// TIA Portal project "PLC_AGV.CENTRAL_V15" (V15)

(* hardware
DEVICE "ET 200S station_1"  ET 200S station
   slot 0: "Rack_0"  Rail
   slot 2: "PLC_AGV.CENTRAL"  IM151-8 PN/DP CPU  6ES7 151-8AB01-0AB0  V3.2
      slot 1: "PROFINET interface_1"  PN-IO
         slot 1: "Port_1"  Port
         slot 2: "Port_2"  Port
         slot 3: "Port_3"  Port
   slot 4: "PM-E 24VDC_1"  PM-E 24VDC  6ES7 138-4CA01-0AA0
   slot 5: "8DI x 24VDC_1"  8DI x 24VDC  6ES7 131-4BF00-0AA0
   slot 6: "8DI x 24VDC_2"  8DI x 24VDC  6ES7 131-4BF00-0AA0
   slot 7: "8DI x 24VDC_3"  8DI x 24VDC  6ES7 131-4BF00-0AA0
   slot 8: "8DI x 24VDC_4"  8DI x 24VDC  6ES7 131-4BF00-0AA0
   slot 9: "8DO x 24VDC / 0.5A_1"  8DO x 24VDC / 0.5A  6ES7 132-4BF00-0AA0
   slot 10: "8DO x 24VDC / 0.5A_2"  8DO x 24VDC / 0.5A  6ES7 132-4BF00-0AA0
   slot 11: "8DO x 24VDC / 0.5A_3"  8DO x 24VDC / 0.5A  6ES7 132-4BF00-0AA0
   slot 12: "8DO x 24VDC / 0.5A_4"  8DO x 24VDC / 0.5A  6ES7 132-4BF00-0AA0
*)

// ===== PLC "PLC_AGV.CENTRAL"  IM151-8 PN/DP CPU =====

VAR_GLOBAL   // PLC tag table "Default tag table"
   "HORN" AT %Q5.0 : Bool;
   "LAMP1" AT %Q5.2 : Bool;
   "LAMP2" AT %Q5.4 : Bool;
   "LAMP3" AT %Q5.6 : Bool;
   "DI.Start_D1" AT %I3.0 : Bool;
   "DI.Stop_D1" AT %I3.1 : Bool;
   "DI.Start_D2" AT %I3.2 : Bool;
   "DI.Stop_D2" AT %I3.3 : Bool;
   "DI.Start_D3" AT %I3.4 : Bool;
   "DI.Stop_D3" AT %I3.5 : Bool;
   "DI.Start_D4" AT %I3.6 : Bool;
   "DI.Stop_D4" AT %I3.7 : Bool;
   "DI_BufferScanner" AT %I4.0 : Bool;   // Scanner to check buffer height
   "DO_GreenLight" AT %Q6.0 : Bool;   // Green light to indicate buffer height
   "DO_RedLight" AT %Q6.1 : Bool;   // Red light - buffer overheight
   "DO_BufferBuzzer" AT %Q6.2 : Bool;   // Buzzer buffer overheight
   "Always_True" AT %M10.0 : Bool;
   "Always_False" AT %M10.1 : Bool;
END_VAR

VAR_GLOBAL CONSTANT   // PLC tag table "Default tag table"
   "QTY.AGV" : Int := 7;
   "MAX.STATIONS" : Int := 8;
END_VAR

VAR_GLOBAL   // PLC tag table "ClockMemory"
   "CM_0.1s" AT %M0.0 : Bool;
   "CM_0.2s" AT %M0.1 : Bool;
   "CM_0.4s" AT %M0.2 : Bool;
   "CM_0.5s" AT %M0.3 : Bool;
   "CM_0.8s" AT %M0.4 : Bool;
   "CM_1s" AT %M0.5 : Bool;
   "CM_1.6s" AT %M0.6 : Bool;
   "CM_2s" AT %M0.7 : Bool;
END_VAR

VAR_GLOBAL   // PLC tag table "IO tag table"
   "STATION1.STOP" AT %I1.0 : Bool;
   "STATION1.RUN" AT %I1.1 : Bool;
   "STATION2.STOP" AT %I1.2 : Bool;
   "STATION2.RUN" AT %I1.3 : Bool;
   "STATION3.STOP" AT %I1.4 : Bool;
   "STATION3.RUN" AT %I1.5 : Bool;
   "STATION4.STOP" AT %I1.6 : Bool;
   "STATION4.RUN" AT %I1.7 : Bool;
   "STATION5.STOP" AT %I2.0 : Bool;
   "STATION5.RUN" AT %I2.1 : Bool;
   "STATION6.STOP" AT %I2.2 : Bool;
   "STATION6.RUN" AT %I2.3 : Bool;
END_VAR

VAR_GLOBAL   // PLC tag table "MemoriasTakt"
   "Me_PararLinha" AT %M20.0 : Bool;
   "Me_Emergencia" AT %M20.1 : Bool;
   "Me_EmTurno" AT %M20.2 : Bool;
   "Me_ResetTakt" AT %M20.3 : Bool;
   "Me_ParadaProgramada" AT %M20.4 : Bool;
   "Me_PararLinhaAgv" AT %M20.5 : Bool;
   "Ret_Val" AT %MW2 : Int;
   "Error" AT %M1.0 : Bool;
   "Statuts" AT %MW4 : Word;
   "C_Conect" AT %M1.1 : Bool;
   "C_Status" AT %MW6 : Word;
END_VAR

TYPE "Agv.Database"
   STRUCT
      Emergencia : Bool;   // Botao de Emergecencia
      Warning : Bool;   // Area de Warning do Scanner
      Safety : Bool;   // Area de Safety do Scanner
      ConectarTakt : Bool;   // 0 - Desconectado / 1 - Conectado
      Rodando : Bool;
      Falha : Bool;
      AutomaticoManual : Byte;   // 1 - Manual / 2 - Automatico
      VelocidadeAtual : Int;   // Velocidade Atual
      Posto : Byte;   // Posto em que o AGV está
      Comando : Byte;   // Ultimo comando
      Velocidade : Byte;   // Velocidade Setada
      Processo : Byte;   // 1 - Ecu / 2 - SKD
      "Erros.Agv" : Byte;   // 0 á 256, cada numero um erro. 1 - Tudo Ok
      "Erros.Pgv" : Byte;   // 0 á 256, cada numero um erro. 1 - Tudo Ok
      "Erros.Rfid" : Byte;   // 0 á 256, cada numero um erro. 1 - Tudo Ok
      "Erros.MotorPasso" : Byte;   // 0 á 256, cada numero um erro. 1 - Tudo Ok
      "Erros.IOLink" : Byte;   // 0 á 256, cada numero um erro. 1 - Tudo Ok
      "Erros.Comunicacao" : Byte;   // 0 á 256, cada numero um erro. 1 - Tudo Ok
      Reservado : Byte;   // Reservado
      Reservado_1 : Byte;   // Reservado
      Reservado_2 : Byte;   // Reservado
      Reservado_3 : Byte;   // Reservado
      Reservado_4 : Byte;   // Reservado
      Reservado_5 : Byte;   // Reservado
      Reservado_6 : Byte;   // Reservado
      Reservado_7 : Byte;   // Reservado
      Reservado_8 : Byte;   // Reservado
   END_STRUCT;
END_TYPE

TYPE "Takt.Database"
   STRUCT
      EmergenciaECU : Bool;   // Emergencia
      EmergenciaSKD : Bool;   // Emergencia
      StartAgvECU : Bool;   // Start by takt
      StopAgvECU : Bool;   // Stop by takt
      StartAgvSKD : Bool;   // Start by takt
      StopAgvSKD : Bool;   // Stop by takt
      WatchDog : Bool;   // WatchDog
      TOD : Time_Of_Day;   // Time of day
   END_STRUCT;
END_TYPE

TYPE "Scada.Datebase"
   STRUCT
      Turnos : Struct
         Inicio : Array[0..2] of Time_Of_Day;
         Fim : Array[0..2] of Time_Of_Day;
      END_STRUCT;
      Paradas_Programadas : Struct
         Inicio : Array[0..5] of Time_Of_Day;
         Fim : Array[0..5] of Time_Of_Day;
      END_STRUCT;
      Dias_Da_Semana : Array[0..6] of Bool;
      ParametrosTakt : Array[0..2] of Struct
         Tempo_Takt : Int;
         ObjetivoTurno : Int;
      END_STRUCT;
      DiaDaSemana : Int;
   END_STRUCT;
   // // Dias_Da_Semana[0] : Segunda-Feira
   // // Dias_Da_Semana[1] : Terça-Feira
   // // Dias_Da_Semana[2] : Quarta-Feira
   // // Dias_Da_Semana[3] : Quinta-Feira
   // // Dias_Da_Semana[4] : Sexta-Feira
   // // Dias_Da_Semana[5] : Sabado
   // // Dias_Da_Semana[6] : Domingo
   // // ParametrosTakt[0] : Parametros do Takt do 1 turno
   // // ParametrosTakt[1] : Parametros do Takt do 2 turno
   // // ParametrosTakt[2] : Parametros do Takt do 3 turno
   // // Turnos.Inicio[0] : Incio 1 Turno
   // // Turnos.Inicio[1] : Incio 2 Turno
   // // Turnos.Inicio[2] : Incio 3 Turno
   // // Turnos.Fim[0] : Fim 1 Turno
   // // Turnos.Fim[1] : Fim 2 Turno
   // // Turnos.Fim[2] : Fim 3 Turno
   // // Paradas_Programadas.Inicio[0] : Inicio Parada Programada 1
   // // Paradas_Programadas.Inicio[1] : Inicio Parada Programada 2
   // // Paradas_Programadas.Fim[0] : Fim Parada Programada 1
   // // Paradas_Programadas.Inicio[2] : Inicio Parada Programada 3
   // // Paradas_Programadas.Inicio[3] : Inicio Parada Programada 4
   // // Paradas_Programadas.Inicio[4] : Inicio Parada Programada 5
   // // Paradas_Programadas.Inicio[5] : Inicio Parada Programada 6
   // // Paradas_Programadas.Fim[1] : Fim Parada Programada 2
   // // Paradas_Programadas.Fim[2] : Fim Parada Programada 3
   // // Paradas_Programadas.Fim[3] : Fim Parada Programada 4
   // // Paradas_Programadas.Fim[4] : Fim Parada Programada 5
   // // Paradas_Programadas.Fim[5] : Fim Parada Programada 6
END_TYPE

TYPE "UltimasParadas"
   STRUCT
      NumeroPosto : Int;
      InicioParada : Time_Of_Day;
      FimParada : Time_Of_Day;
      DiaDaParada : Date;
   END_STRUCT;
END_TYPE

TYPE "Central.Database"
   STRUCT
      Dados_Agv : Array[0..12] of "Agv.Database";
      Dados_Takt : Struct
         Tempo_Takt : DInt;
         Tempo_StopTime : DInt;
         Objetivo : Int;
         Atual : Int;
         TempoParada : DInt;
         Andons : Array[0..8] of Bool;
      END_STRUCT;
      Dados_Paradas : Array[0..20] of "UltimasParadas";
   END_STRUCT;
END_TYPE

// folder: 01_Takt/02_DB

DATA_BLOCK "DB100_LogicaTaktEcu"   // DB100
{ S7_Optimized_Access := 'FALSE' }
AUTHOR : ssbjvq
VERSION : 0.1
// stored: InstanceOfName FB100_LogicaTaktEcu
"FB100_LogicaTaktEcu"
BEGIN
END_DATA_BLOCK

DATA_BLOCK "DB101_SinaisEmTurno"   // DB101
{ S7_Optimized_Access := 'FALSE' }
VERSION : 0.1
// stored: InstanceOfName FB101_SinaisEmTurno
"FB101_SinaisEmTurno"
BEGIN
END_DATA_BLOCK

DATA_BLOCK "DB102_SinaisDeAndons"   // DB102
{ S7_Optimized_Access := 'FALSE' }
VERSION : 0.1
// stored: InstanceOfName FB102_SinaisDeAndons
"FB102_SinaisDeAndons"
BEGIN
END_DATA_BLOCK

DATA_BLOCK "DB103_AndonsAgvs"   // DB103
{ S7_Optimized_Access := 'FALSE' }
VERSION : 0.1
// stored: InstanceOfName FB103_AndonsAgvs
"FB103_AndonsAgvs"
BEGIN
END_DATA_BLOCK

// folder: 02_Comunicação/02_DB

DATA_BLOCK "DB200_TaktToAgv"   // DB200
TITLE = DB1_TaktToAgv
{ S7_Optimized_Access := 'FALSE' }
AUTHOR : ssbjvq
VERSION : 0.1
// DB1_TaktToAgv
   VAR
      Dados : "Takt.Database";
   END_VAR
BEGIN
   Dados.WatchDog := TRUE;
END_DATA_BLOCK

DATA_BLOCK "DB201_Comunicação"   // DB201
{ S7_Optimized_Access := 'FALSE' }
AUTHOR : ssbjvq
VERSION : 0.1
// stored: InstanceOfName FB201_Comunicação
"FB201_Comunicação"
BEGIN
END_DATA_BLOCK

// folder: 03_Scada

DATA_BLOCK "DB300_ScadaToCentral"   // DB300
TITLE = DB300_MestreToCentral
{ S7_Optimized_Access := 'FALSE' }
VERSION : 0.1
// DB300_MestreToCentral
   VAR
      Data : "Scada.Datebase";
   END_VAR
BEGIN
   Data.Turnos.Inicio[0] := TOD#08:00:00;
   Data.Turnos.Inicio[1] := TOD#00:00:00;
   Data.Turnos.Inicio[2] := TOD#00:00:00;
   Data.Turnos.Fim[0] := TOD#15:55:00;
   Data.Turnos.Fim[1] := TOD#00:00:00;
   Data.Turnos.Fim[2] := TOD#00:00:00;
   Data.Dias_Da_Semana[0] := TRUE;
   Data.Dias_Da_Semana[1] := TRUE;
   Data.Dias_Da_Semana[2] := TRUE;
   Data.Dias_Da_Semana[3] := TRUE;
   Data.Dias_Da_Semana[4] := TRUE;
   Data.ParametrosTakt[0].Tempo_Takt := 600;
   Data.ParametrosTakt[0].ObjetivoTurno := 48;
   Data.ParametrosTakt[1].Tempo_Takt := 600;
   Data.ParametrosTakt[1].ObjetivoTurno := 48;
   Data.ParametrosTakt[2].Tempo_Takt := 600;
   Data.ParametrosTakt[2].ObjetivoTurno := 48;
   Data.DiaDaSemana := 2;
   Data.Paradas_Programadas.Fim[0] := TOD#12:15:00;
   Data.Paradas_Programadas.Inicio[0] := TOD#11:15:00;
END_DATA_BLOCK

DATA_BLOCK "DB301_CentralToScada"   // DB301
TITLE = DB301_CentralToScada
{ S7_Optimized_Access := 'FALSE' }
VERSION : 0.1
// DB301_CentralToScada
   VAR
      Data : "Central.Database";
   END_VAR
BEGIN
END_DATA_BLOCK

// folder: 04_Services/02_DB

DATA_BLOCK "FB1000_Clock_DB"   // DB1
{ S7_Optimized_Access := 'FALSE' }
VERSION : 0.1
// stored: InstanceOfName FB1000_Clock
"FB1000_Clock"
BEGIN
END_DATA_BLOCK

// folder: (top level)

ORGANIZATION_BLOCK "Main"   // OB1, LAD
TITLE = "Main Program Sweep (Cycle)"
{ S7_Optimized_Access := 'FALSE' }
VERSION : 0.1
   VAR_TEMP
      OB1_EV_CLASS : Byte;   // Bits 0-3 = 1 (Coming event), Bits 4-7 = 1 (Event class 1)
      OB1_SCAN_1 : Byte;   // 1 (Cold restart scan 1 of OB 1), 3 (Scan 2-n of OB 1)
      OB1_PRIORITY : Byte;   // Priority of OB Execution
      OB1_OB_NUMBR : Byte;   // 1 (Organization block 1, OB1)
      OB1_RESERVED_1 : Byte;   // Reserved for system
      OB1_RESERVED_2 : Byte;   // Reserved for system
      OB1_PREV_CYCLE : Int;   // Cycle time of previous OB1 scan (milliseconds)
      OB1_MIN_CYCLE : Int;   // Minimum cycle time of OB1 (milliseconds)
      OB1_MAX_CYCLE : Int;   // Maximum cycle time of OB1 (milliseconds)
      OB1_DATE_TIME : Date_And_Time;   // Date and time OB1 started
   END_VAR
BEGIN

REGION Network 1: Filtro dos botões de Andon
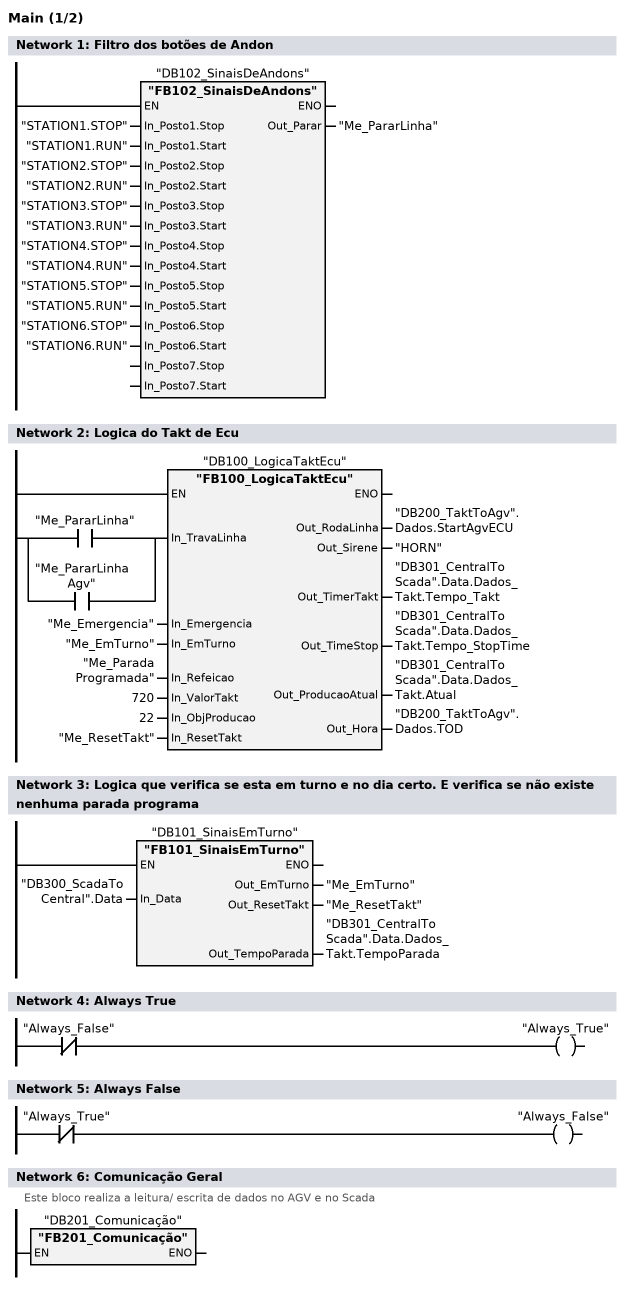
   RUNG wire#powerrail
      "DB102_SinaisDeAndons"("In_Posto1.Stop" := "STATION1.STOP", "In_Posto1.Start" := "STATION1.RUN", "In_Posto2.Stop" := "STATION2.STOP", "In_Posto2.Start" := "STATION2.RUN", "In_Posto3.Stop" := "STATION3.STOP", "In_Posto3.Start" := "STATION3.RUN", "In_Posto4.Stop" := "STATION4.STOP", "In_Posto4.Start" := "STATION4.RUN", "In_Posto5.Stop" := "STATION5.STOP", "In_Posto5.Start" := "STATION5.RUN", "In_Posto6.Stop" := "STATION6.STOP", "In_Posto6.Start" := "STATION6.RUN", "In_Posto7.Stop" :=, "In_Posto7.Start" :=, Out_Parar => "Me_PararLinha")
   END_RUNG
   // the same network as SCL:
   "DB102_SinaisDeAndons"("In_Posto1.Stop" := "STATION1.STOP",   // "FB102_SinaisDeAndons"
                          "In_Posto1.Start" := "STATION1.RUN",
                          "In_Posto2.Stop" := "STATION2.STOP",
                          "In_Posto2.Start" := "STATION2.RUN",
                          "In_Posto3.Stop" := "STATION3.STOP",
                          "In_Posto3.Start" := "STATION3.RUN",
                          "In_Posto4.Stop" := "STATION4.STOP",
                          "In_Posto4.Start" := "STATION4.RUN",
                          "In_Posto5.Stop" := "STATION5.STOP",
                          "In_Posto5.Start" := "STATION5.RUN",
                          "In_Posto6.Stop" := "STATION6.STOP",
                          "In_Posto6.Start" := "STATION6.RUN",
                          Out_Parar => "Me_PararLinha");
END_REGION

REGION Network 2: Logica do Takt de Ecu
   RUNG wire#powerrail
      "DB100_LogicaTaktEcu"(In_TravaLinha := wire#w1, In_Emergencia := "Me_Emergencia", In_EmTurno := "Me_EmTurno", In_Refeicao := "Me_ParadaProgramada", In_ValorTakt := 720, In_ObjProducao := 22, In_ResetTakt := "Me_ResetTakt", Out_RodaLinha => "DB200_TaktToAgv".Dados.StartAgvECU, Out_Sirene => "HORN", Out_TimerTakt => "DB301_CentralToScada".Data.Dados_Takt.Tempo_Takt, Out_TimeStop => "DB301_CentralToScada".Data.Dados_Takt.Tempo_StopTime, Out_ProducaoAtual => "DB301_CentralToScada".Data.Dados_Takt.Atual, Out_Hora => "DB200_TaktToAgv".Dados.TOD)
   END_RUNG
   RUNG wire#powerrail
      Contact( "Me_PararLinha" )
   END_RUNG wire#w1
   RUNG wire#powerrail
      Contact( "Me_PararLinhaAgv" )
   END_RUNG wire#w1
   // the same network as SCL:
   "DB100_LogicaTaktEcu"(In_TravaLinha := "Me_PararLinha" OR "Me_PararLinhaAgv",   // "FB100_LogicaTaktEcu"
                         In_Emergencia := "Me_Emergencia",
                         In_EmTurno := "Me_EmTurno",
                         In_Refeicao := "Me_ParadaProgramada",
                         In_ValorTakt := 720,
                         In_ObjProducao := 22,
                         In_ResetTakt := "Me_ResetTakt",
                         Out_RodaLinha => "DB200_TaktToAgv".Dados.StartAgvECU,
                         Out_Sirene => "HORN",
                         Out_TimerTakt => "DB301_CentralToScada".Data.Dados_Takt.Tempo_Takt,
                         Out_TimeStop => "DB301_CentralToScada".Data.Dados_Takt.Tempo_StopTime,
                         Out_ProducaoAtual => "DB301_CentralToScada".Data.Dados_Takt.Atual,
                         Out_Hora => "DB200_TaktToAgv".Dados.TOD);
END_REGION

REGION Network 3: Logica que verifica se esta em turno e no dia certo. E verifica se não existe nenhuma parada programa
   RUNG wire#powerrail
      "DB101_SinaisEmTurno"(In_Data := "DB300_ScadaToCentral".Data, Out_EmTurno => "Me_EmTurno", Out_ResetTakt => "Me_ResetTakt", Out_TempoParada => "DB301_CentralToScada".Data.Dados_Takt.TempoParada)
   END_RUNG
   // the same network as SCL:
   "DB101_SinaisEmTurno"(In_Data := "DB300_ScadaToCentral".Data,   // "FB101_SinaisEmTurno"
                         Out_EmTurno => "Me_EmTurno",
                         Out_ResetTakt => "Me_ResetTakt",
                         Out_TempoParada => "DB301_CentralToScada".Data.Dados_Takt.TempoParada);
END_REGION

REGION Network 4: Always True
   RUNG wire#powerrail
      I_Contact( "Always_False" )
      Coil( "Always_True" )
   END_RUNG
   // the same network as SCL:
   "Always_True" := NOT "Always_False";
END_REGION

REGION Network 5: Always False
   RUNG wire#powerrail
      I_Contact( "Always_True" )
      Coil( "Always_False" )
   END_RUNG
   // the same network as SCL:
   "Always_False" := NOT "Always_True";
END_REGION

REGION Network 6: Comunicação Geral
   // Este bloco realiza a leitura/ escrita de dados no AGV e no Scada
   RUNG wire#powerrail
      "DB201_Comunicação"()
   END_RUNG
   // the same network as SCL:
   "DB201_Comunicação"();   // "FB201_Comunicação"
END_REGION

REGION Network 7: Sinais de Andon dos Agvs
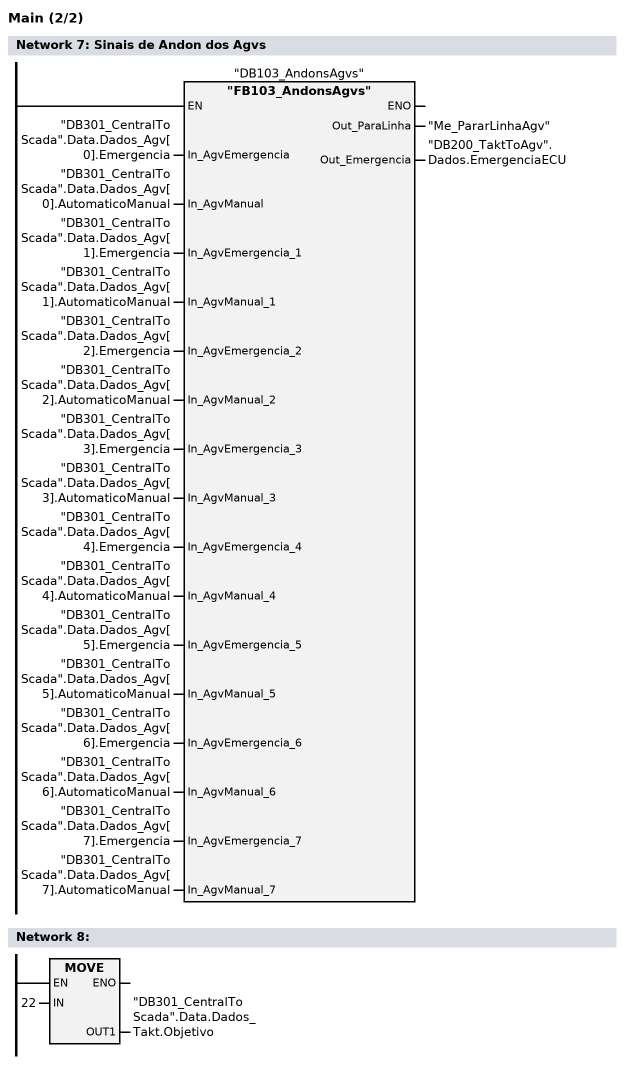
   RUNG wire#powerrail
      "DB103_AndonsAgvs"(In_AgvEmergencia := "DB301_CentralToScada".Data.Dados_Agv[0].Emergencia, In_AgvManual := "DB301_CentralToScada".Data.Dados_Agv[0].AutomaticoManual, In_AgvEmergencia_1 := "DB301_CentralToScada".Data.Dados_Agv[1].Emergencia, In_AgvManual_1 := "DB301_CentralToScada".Data.Dados_Agv[1].AutomaticoManual, In_AgvEmergencia_2 := "DB301_CentralToScada".Data.Dados_Agv[2].Emergencia, In_AgvManual_2 := "DB301_CentralToScada".Data.Dados_Agv[2].AutomaticoManual, In_AgvEmergencia_3 := "DB301_CentralToScada".Data.Dados_Agv[3].Emergencia, In_AgvManual_3 := "DB301_CentralToScada".Data.Dados_Agv[3].AutomaticoManual, In_AgvEmergencia_4 := "DB301_CentralToScada".Data.Dados_Agv[4].Emergencia, In_AgvManual_4 := "DB301_CentralToScada".Data.Dados_Agv[4].AutomaticoManual, In_AgvEmergencia_5 := "DB301_CentralToScada".Data.Dados_Agv[5].Emergencia, In_AgvManual_5 := "DB301_CentralToScada".Data.Dados_Agv[5].AutomaticoManual, In_AgvEmergencia_6 := "DB301_CentralToScada".Data.Dados_Agv[6].Emergencia, In_AgvManual_6 := "DB301_CentralToScada".Data.Dados_Agv[6].AutomaticoManual, In_AgvEmergencia_7 := "DB301_CentralToScada".Data.Dados_Agv[7].Emergencia, In_AgvManual_7 := "DB301_CentralToScada".Data.Dados_Agv[7].AutomaticoManual, Out_ParaLinha => "Me_PararLinhaAgv", Out_Emergencia => "DB200_TaktToAgv".Dados.EmergenciaECU)
   END_RUNG
   // the same network as SCL:
   "DB103_AndonsAgvs"(In_AgvEmergencia := "DB301_CentralToScada".Data.Dados_Agv[0].Emergencia,   // "FB103_AndonsAgvs"
                      In_AgvManual := "DB301_CentralToScada".Data.Dados_Agv[0].AutomaticoManual,
                      In_AgvEmergencia_1 := "DB301_CentralToScada".Data.Dados_Agv[1].Emergencia,
                      In_AgvManual_1 := "DB301_CentralToScada".Data.Dados_Agv[1].AutomaticoManual,
                      In_AgvEmergencia_2 := "DB301_CentralToScada".Data.Dados_Agv[2].Emergencia,
                      In_AgvManual_2 := "DB301_CentralToScada".Data.Dados_Agv[2].AutomaticoManual,
                      In_AgvEmergencia_3 := "DB301_CentralToScada".Data.Dados_Agv[3].Emergencia,
                      In_AgvManual_3 := "DB301_CentralToScada".Data.Dados_Agv[3].AutomaticoManual,
                      In_AgvEmergencia_4 := "DB301_CentralToScada".Data.Dados_Agv[4].Emergencia,
                      In_AgvManual_4 := "DB301_CentralToScada".Data.Dados_Agv[4].AutomaticoManual,
                      In_AgvEmergencia_5 := "DB301_CentralToScada".Data.Dados_Agv[5].Emergencia,
                      In_AgvManual_5 := "DB301_CentralToScada".Data.Dados_Agv[5].AutomaticoManual,
                      In_AgvEmergencia_6 := "DB301_CentralToScada".Data.Dados_Agv[6].Emergencia,
                      In_AgvManual_6 := "DB301_CentralToScada".Data.Dados_Agv[6].AutomaticoManual,
                      In_AgvEmergencia_7 := "DB301_CentralToScada".Data.Dados_Agv[7].Emergencia,
                      In_AgvManual_7 := "DB301_CentralToScada".Data.Dados_Agv[7].AutomaticoManual,
                      Out_ParaLinha => "Me_PararLinhaAgv",
                      Out_Emergencia => "DB200_TaktToAgv".Dados.EmergenciaECU);
END_REGION

REGION Network 8
   RUNG wire#powerrail
      { S7_GenerateENO := "TRUE" } Move(in := 22, out1 => "DB301_CentralToScada".Data.Dados_Takt.Objetivo)
   END_RUNG
   // the same network as SCL:
   "DB301_CentralToScada".Data.Dados_Takt.Objetivo := 22;
END_REGION
END_ORGANIZATION_BLOCK

// folder: 01_Takt/01_FB

FUNCTION_BLOCK "FB100_LogicaTaktEcu"   // FB100, SCL
TITLE = FB100_LogicaTaktEcu
{ S7_Optimized_Access := 'FALSE' }
AUTHOR : ssbjvq
VERSION : 0.1
// FB100_LogicaTaktEcu
   VAR_INPUT
      In_TravaLinha : Bool;   // Input dos andons. True - Para Linha/ False - Tudo Ok!
      In_Emergencia : Bool;   // Inout de Emergencia. True - Acionado/ False - Desacionado
      In_EmTurno : Bool;   // Input dos Em turno. True - Linha em turno/ False - Fora do turno
      In_Refeicao : Bool;   // Input de Pause Programada. True - Em horario de parada / False - Fora do horario de parada
      In_ValorTakt : Int;   // Input do valor do Takt
      In_ObjProducao : Int;   // Input do Objetivo de producao
      In_ResetTakt : Bool;   // Sinal que reseta o Stop Time
   END_VAR
   VAR_OUTPUT
      Out_RodaLinha : Bool;   // Out Roda Linha
      Out_Sirene : Bool;   // Out Sirene
      Out_TimerTakt : DInt;   // Out Tempo Takt
      Out_TimeStop : DInt;   // Out Tempo Stop time
      Out_ProducaoAtual : Int;   // Out Contagem Producao
      Out_Hora : Time_Of_Day;
   END_VAR
   VAR
      S_TudoOk : Bool;   // Inicia a contagem do Takt
      S_ResetTakt : Bool;   // Reseta o Takt
      S_StopLinha : Bool;   // Inicia a contagem do Stop time
      S_Reset_Stop : Bool;   // Reseta o Stop Time E Contagem Producao
      S_TaktTimeAtual : DInt;   // Tempo Atual do Takt ( Regressivo)
      Contador_Takt : CTU;   // Contador do Takt
      Contador_StopTime : CTU;   // Contador do Stop Time
      Contador_Producao : CTU;   // Contador de Producao
      Start_Takt : TP;
      S_DateTime : Date_And_Time;
      S_ResetAllTakt : Bool;
   END_VAR
   VAR_TEMP
      Err : Int;
   END_VAR
BEGIN
   (*
    BLOCO DESENVOLVIDO POR SSBJVQ R.4946
    BLOCO DO TAKT
   *)

   REGION Logica Takt
       IF #In_ResetTakt THEN
           #S_ResetTakt := 1;
           #S_TudoOk := 0;
           #S_StopLinha := 0;
           #S_ResetTakt := 0;
           #S_Reset_Stop := 1;
       END_IF;
       // Verifica as condições para acionar a contagem do Takt
       IF (#In_EmTurno AND NOT #In_Refeicao AND
           (#Contador_Takt.CV < #In_ValorTakt) AND (#Contador_Producao.CV < #In_ObjProducao)) AND NOT #In_ResetTakt THEN
           #S_TudoOk := 1;
           #S_StopLinha := 0;
           #S_ResetTakt := 0;
           #S_Reset_Stop := 0;

           // Verifica as condições para acionar a contagem do Stop Time
       ELSIF ((#In_Emergencia OR #In_TravaLinha) AND (#Contador_Takt.CV = #In_ValorTakt)
           AND (#Contador_Producao.CV < #In_ObjProducao) AND #In_EmTurno) AND NOT #In_ResetTakt THEN
           #S_TudoOk := 0;
           #S_StopLinha := 1;
           #S_ResetTakt := 0;
           #S_Reset_Stop := 0;
           // Verifica as condições para acionar o Reset Takt
       ELSIF (#In_EmTurno
           AND NOT #In_Refeicao AND NOT #In_Emergencia
           AND NOT #In_TravaLinha AND (#Contador_Takt.CV = #In_ValorTakt) AND #Contador_Takt.Q)AND NOT #In_ResetTakt THEN
           #S_ResetTakt := 1;
           // Verifica se esta em parada programada
       ELSIF NOT #In_EmTurno AND #In_Refeicao AND NOT #In_ResetTakt THEN
           #S_TudoOk := 0;
           #S_StopLinha := 0;
           #S_Reset_Stop := 0;
           #S_ResetTakt := 0;
       // Verifica as condições para acionar o Reset Stop Time
       ELSIF #In_ResetTakt THEN
           #S_Reset_Stop := 1;
           #S_TudoOk := 0;
           #S_StopLinha := 0;
           #S_ResetTakt := 1;
       ELSE
           #S_TudoOk := 0;
           #S_StopLinha := 0;
           #S_Reset_Stop := 0;
           #S_ResetTakt := 0;
       END_IF;

       #Err := RD_SYS_T(#S_DateTime);
   END_REGION

   IF DT_TO_TOD(#S_DateTime) >= TOD#07:00:00 AND  DT_TO_TOD(#S_DateTime)<= TOD#07:01:00
       OR DT_TO_TOD(#S_DateTime) >= TOD#17:00:00 AND  DT_TO_TOD(#S_DateTime)<= TOD#17:01:00
       OR DT_TO_TOD(#S_DateTime) >= TOD#00:00:00 AND  DT_TO_TOD(#S_DateTime)<= TOD#00:01:00 THEN
       #S_ResetAllTakt := 1;
   ELSE
       #S_ResetAllTakt := 0;
   END_IF;


   // Contém os contadores do TAKT, Stop Time e Producao
   REGION Contadores

       #Contador_Takt(CU := #S_TudoOk AND "CM_1s",
                      R := #S_ResetTakt OR #In_ResetTakt OR #S_ResetAllTakt ,
                      PV := #In_ValorTakt);
       #Contador_StopTime(CU := #S_StopLinha AND "CM_1s" ,
                          R :=  #S_Reset_Stop OR #In_ResetTakt OR #S_ResetAllTakt
                          ,
                          PV := 32747);
       #Contador_Producao(CU := #Contador_Takt.Q ,
                          R := #S_Reset_Stop OR #In_ResetTakt OR #S_ResetAllTakt  ,
                          PV := #In_ObjProducao);
       // Timer que dá o start nos AGVs e mantém 'startado' por 10s
       #Start_Takt(IN:=NOT #In_TravaLinha AND
                   NOT #In_Emergencia AND
                   NOT #In_Refeicao AND 
                   #In_EmTurno AND (#S_TaktTimeAtual <= 0) ,
                   PT:=T#10s);


   END_REGION


   //Joga as memorias nas saidas do bloco
   REGION Saidas
       #Out_RodaLinha := #Start_Takt.Q;
       #S_TaktTimeAtual := INT_TO_DINT(#Contador_Takt.CV);
       #Out_TimerTakt := (INT_TO_DINT(#In_ValorTakt) - #S_TaktTimeAtual);
       #Out_TimeStop := INT_TO_DINT(#Contador_StopTime.CV);
       #Out_ProducaoAtual := #Contador_Producao.CV;
       #Out_Sirene := ((#Out_TimerTakt > 1 AND #Out_TimerTakt < 5)OR (#Out_TimerTakt > 25  AND #Out_TimerTakt < 30)OR(#Start_Takt.ET > T#100ms AND  #Start_Takt.ET < T#5s )) AND "CM_0.5s" ;
       #Out_Hora := DT_TO_TOD(#S_DateTime);
   END_REGION
END_FUNCTION_BLOCK

FUNCTION_BLOCK "FB101_SinaisEmTurno"   // FB101, SCL
TITLE = FB101_SinaisDeAndons
{ S7_Optimized_Access := 'FALSE' }
VERSION : 0.1
// FB101_SinaisDeAndons
   VAR_INPUT
      In_Data : "Scada.Datebase";   // Dados vindos do Scada IT
   END_VAR
   VAR_OUTPUT
      Out_EmTurno : Bool;   // Memoria que verifica se está em turno
      Out_ResetTakt : Bool;   // Memoria para resetar o takt/stop time
      Out_TempoParada : DInt;   // Valor que está falta para o turno iniciar
   END_VAR
   VAR
      S_Date_Time : Date_And_Time;
      S_Time : Time_Of_Day;
      S_EmTurno : Array[0..2] of Bool;
      S_ParadaProgramada : Array[0..5] of Bool;
      S_DiaDaSemana : Array[0..6] of Bool;
      S_ResetTakt : Array[0..2] of Bool;
      S_Turno : Bool;
      S_Parada : Bool;
      S_DiaSemana : Bool;
      TP_ResetTakt : TP;
      S_TempoParada : DInt;
      S_TODParada : Time_Of_Day;
   END_VAR
   VAR_TEMP
      Err : Int;
      "Counter" : Int;
      Counter_1 : Int;
      Counter_2 : Int;
   END_VAR
BEGIN
   // Realiza a leitura da hora
   #Err := RD_SYS_T(#S_Date_Time);
   #S_Time := DT_TO_TOD(#S_Date_Time);

   #TP_ResetTakt(IN:=(#S_ResetTakt[0] OR #S_ResetTakt[1] OR #S_ResetTakt[2]),
                 PT:=T#10s);




   // Verifica se esta no horario de produção
   FOR #Counter := 0 TO 2 DO
       IF #S_Time >= #In_Data.Turnos.Inicio[#Counter] AND #S_Time <= #In_Data.Turnos.Fim[#Counter] THEN
           IF #S_Time >= #In_Data.Turnos.Inicio[#Counter] AND #S_Time <= (#In_Data.Turnos.Inicio[#Counter] + t#20S) THEN
               #S_ResetTakt[#Counter] := 1;
           ELSE
               #S_ResetTakt[#Counter] := 0;
               #S_EmTurno[#Counter] := 1;
           END_IF;


       ELSE
           #S_EmTurno[#Counter] := 0;
       END_IF;

   END_FOR;

   // Verifica se existe alguma parada programada
   FOR #Counter_1 := 0 TO 5 DO
       IF #S_Time >= #In_Data.Paradas_Programadas.Inicio[#Counter_1] AND #S_Time <= #In_Data.Paradas_Programadas.Fim[#Counter_1] THEN
           #S_ParadaProgramada[#Counter_1] := 1;
       ELSE
           #S_ParadaProgramada[#Counter_1] := 0;
       END_IF;
   END_FOR;

   // Verifica os dias da Semana
   FOR #Counter_2 := 0 TO 6 DO
       IF #In_Data.Dias_Da_Semana[#Counter_2] THEN
           IF #Counter_2 = #In_Data.DiaDaSemana THEN
               #S_DiaDaSemana[#Counter_2] := 1;
           ELSE
               #S_DiaDaSemana[#Counter_2] := 0;
           END_IF;
       END_IF;
   END_FOR;
   // Centralizador de memorias
   #S_Turno := (#S_EmTurno[0] OR #S_EmTurno[1] OR #S_EmTurno[2]);
   #S_Parada := (#S_ParadaProgramada[0] OR #S_ParadaProgramada[1] OR #S_ParadaProgramada[2] OR #S_ParadaProgramada[3] OR #S_ParadaProgramada[4] OR #S_ParadaProgramada[5]);
   #S_DiaSemana := (#S_DiaDaSemana[0] OR #S_DiaDaSemana[1] OR #S_DiaDaSemana[2] OR #S_DiaDaSemana[3] OR #S_DiaDaSemana[4] OR #S_DiaDaSemana[5] OR #S_DiaDaSemana[6]);

   // Verifica se esta em turno, no dia certo e sem paradas
   IF #S_Turno AND #S_DiaSemana AND NOT #S_Parada THEN
       #Out_EmTurno := 1;
   ELSE
       #Out_EmTurno := 0;
   END_IF;

   // Verifica se está em parada planejada e faz a conta de quanto falta para acabar a parada
   REGION TempoRestante
       IF #S_Parada THEN
           IF #S_ParadaProgramada[0] THEN
               #S_TempoParada := TOD_TO_DINT(#In_Data.Paradas_Programadas.Fim[0]) - TOD_TO_DINT(#S_Time);
               ;
           ELSIF #S_ParadaProgramada[1] THEN
               #S_TempoParada := TOD_TO_DINT(#In_Data.Paradas_Programadas.Fim[1]) - TOD_TO_DINT(#S_Time);

           ELSIF #S_ParadaProgramada[2] THEN
               #S_TempoParada := TOD_TO_DINT(#In_Data.Paradas_Programadas.Fim[2]) - TOD_TO_DINT(#S_Time);
               ;
           ELSIF #S_ParadaProgramada[3] THEN
               #S_TempoParada := TOD_TO_DINT(#In_Data.Paradas_Programadas.Fim[3]) - TOD_TO_DINT(#S_Time);
               ;
           ELSIF #S_ParadaProgramada[4] THEN
               #S_TempoParada := TOD_TO_DINT(#In_Data.Paradas_Programadas.Fim[4]) - TOD_TO_DINT(#S_Time);
               ;
           ELSIF #S_ParadaProgramada[5] THEN
               #S_TempoParada := TOD_TO_DINT(#In_Data.Paradas_Programadas.Fim[5]) - TOD_TO_DINT(#S_Time);
               ;
           END_IF;
       ELSIF NOT #S_Turno THEN
           IF #S_EmTurno[0] THEN
               #S_TempoParada := TOD_TO_DINT(#In_Data.Turnos.Inicio[0]) - TOD_TO_DINT(#S_Time);
           ELSIF #S_EmTurno[1] THEN
               #S_TempoParada := TOD_TO_DINT(#In_Data.Turnos.Inicio[1]) - TOD_TO_DINT(#S_Time);
           ELSIF #S_EmTurno[2] THEN
               #S_TempoParada := TOD_TO_DINT(#In_Data.Turnos.Inicio[2]) - TOD_TO_DINT(#S_Time);
           END_IF;
       ELSE
           #S_TempoParada := 0;
       END_IF;


   END_REGION


   #S_TODParada := DINT_TO_TOD(#S_TempoParada);
   #Out_TempoParada := #S_TempoParada;
   #Out_ResetTakt := #TP_ResetTakt.Q;
END_FUNCTION_BLOCK

FUNCTION_BLOCK "FB102_SinaisDeAndons"   // FB102, LAD
TITLE = FB102_SinaisDeAndons
{ S7_Optimized_Access := 'FALSE' }
VERSION : 0.1
   VAR_INPUT
      "In_Posto1.Stop" : Bool;
      "In_Posto1.Start" : Bool;
      "In_Posto2.Stop" : Bool;
      "In_Posto2.Start" : Bool;
      "In_Posto3.Stop" : Bool;
      "In_Posto3.Start" : Bool;
      "In_Posto4.Stop" : Bool;
      "In_Posto4.Start" : Bool;
      "In_Posto5.Stop" : Bool;
      "In_Posto5.Start" : Bool;
      "In_Posto6.Stop" : Bool;
      "In_Posto6.Start" : Bool;
      "In_Posto7.Stop" : Bool;
      "In_Posto7.Start" : Bool;
   END_VAR
   VAR_OUTPUT
      Out_Parar : Bool;
   END_VAR
   VAR
      S_Postos : Array[0..8] of Bool;
   END_VAR
BEGIN

REGION Network 1: Posto 1
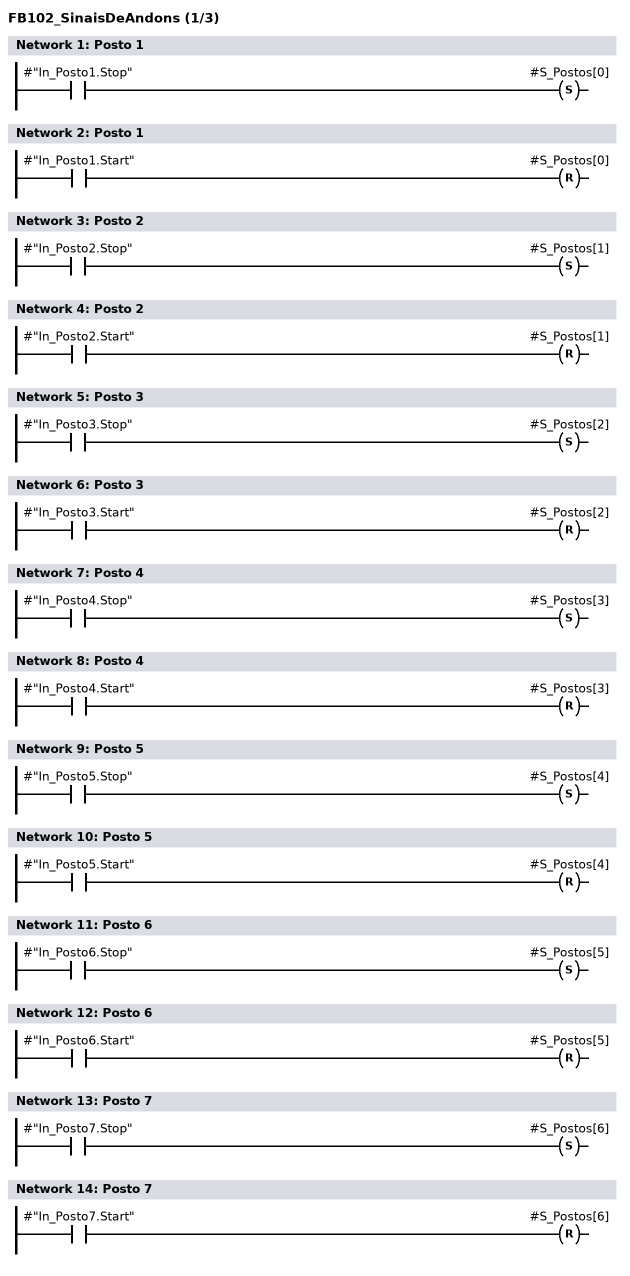
   RUNG wire#powerrail
      Contact( #"In_Posto1.Stop" )
      S_Coil( #S_Postos[0] )
   END_RUNG
   // the same network as SCL:
   IF #"In_Posto1.Stop" THEN #S_Postos[0] := TRUE; END_IF;
END_REGION

REGION Network 2: Posto 1
   RUNG wire#powerrail
      Contact( #"In_Posto1.Start" )
      R_Coil( #S_Postos[0] )
   END_RUNG
   // the same network as SCL:
   IF #"In_Posto1.Start" THEN #S_Postos[0] := FALSE; END_IF;
END_REGION

REGION Network 3: Posto 2
   RUNG wire#powerrail
      Contact( #"In_Posto2.Stop" )
      S_Coil( #S_Postos[1] )
   END_RUNG
   // the same network as SCL:
   IF #"In_Posto2.Stop" THEN #S_Postos[1] := TRUE; END_IF;
END_REGION

REGION Network 4: Posto 2
   RUNG wire#powerrail
      Contact( #"In_Posto2.Start" )
      R_Coil( #S_Postos[1] )
   END_RUNG
   // the same network as SCL:
   IF #"In_Posto2.Start" THEN #S_Postos[1] := FALSE; END_IF;
END_REGION

REGION Network 5: Posto 3
   RUNG wire#powerrail
      Contact( #"In_Posto3.Stop" )
      S_Coil( #S_Postos[2] )
   END_RUNG
   // the same network as SCL:
   IF #"In_Posto3.Stop" THEN #S_Postos[2] := TRUE; END_IF;
END_REGION

REGION Network 6: Posto 3
   RUNG wire#powerrail
      Contact( #"In_Posto3.Start" )
      R_Coil( #S_Postos[2] )
   END_RUNG
   // the same network as SCL:
   IF #"In_Posto3.Start" THEN #S_Postos[2] := FALSE; END_IF;
END_REGION

REGION Network 7: Posto 4
   RUNG wire#powerrail
      Contact( #"In_Posto4.Stop" )
      S_Coil( #S_Postos[3] )
   END_RUNG
   // the same network as SCL:
   IF #"In_Posto4.Stop" THEN #S_Postos[3] := TRUE; END_IF;
END_REGION

REGION Network 8: Posto 4
   RUNG wire#powerrail
      Contact( #"In_Posto4.Start" )
      R_Coil( #S_Postos[3] )
   END_RUNG
   // the same network as SCL:
   IF #"In_Posto4.Start" THEN #S_Postos[3] := FALSE; END_IF;
END_REGION

REGION Network 9: Posto 5
   RUNG wire#powerrail
      Contact( #"In_Posto5.Stop" )
      S_Coil( #S_Postos[4] )
   END_RUNG
   // the same network as SCL:
   IF #"In_Posto5.Stop" THEN #S_Postos[4] := TRUE; END_IF;
END_REGION

REGION Network 10: Posto 5
   RUNG wire#powerrail
      Contact( #"In_Posto5.Start" )
      R_Coil( #S_Postos[4] )
   END_RUNG
   // the same network as SCL:
   IF #"In_Posto5.Start" THEN #S_Postos[4] := FALSE; END_IF;
END_REGION

REGION Network 11: Posto 6
   RUNG wire#powerrail
      Contact( #"In_Posto6.Stop" )
      S_Coil( #S_Postos[5] )
   END_RUNG
   // the same network as SCL:
   IF #"In_Posto6.Stop" THEN #S_Postos[5] := TRUE; END_IF;
END_REGION

REGION Network 12: Posto 6
   RUNG wire#powerrail
      Contact( #"In_Posto6.Start" )
      R_Coil( #S_Postos[5] )
   END_RUNG
   // the same network as SCL:
   IF #"In_Posto6.Start" THEN #S_Postos[5] := FALSE; END_IF;
END_REGION

REGION Network 13: Posto 7
   RUNG wire#powerrail
      Contact( #"In_Posto7.Stop" )
      S_Coil( #S_Postos[6] )
   END_RUNG
   // the same network as SCL:
   IF #"In_Posto7.Stop" THEN #S_Postos[6] := TRUE; END_IF;
END_REGION

REGION Network 14: Posto 7
   RUNG wire#powerrail
      Contact( #"In_Posto7.Start" )
      R_Coil( #S_Postos[6] )
   END_RUNG
   // the same network as SCL:
   IF #"In_Posto7.Start" THEN #S_Postos[6] := FALSE; END_IF;
END_REGION

REGION Network 15: Parar Linha
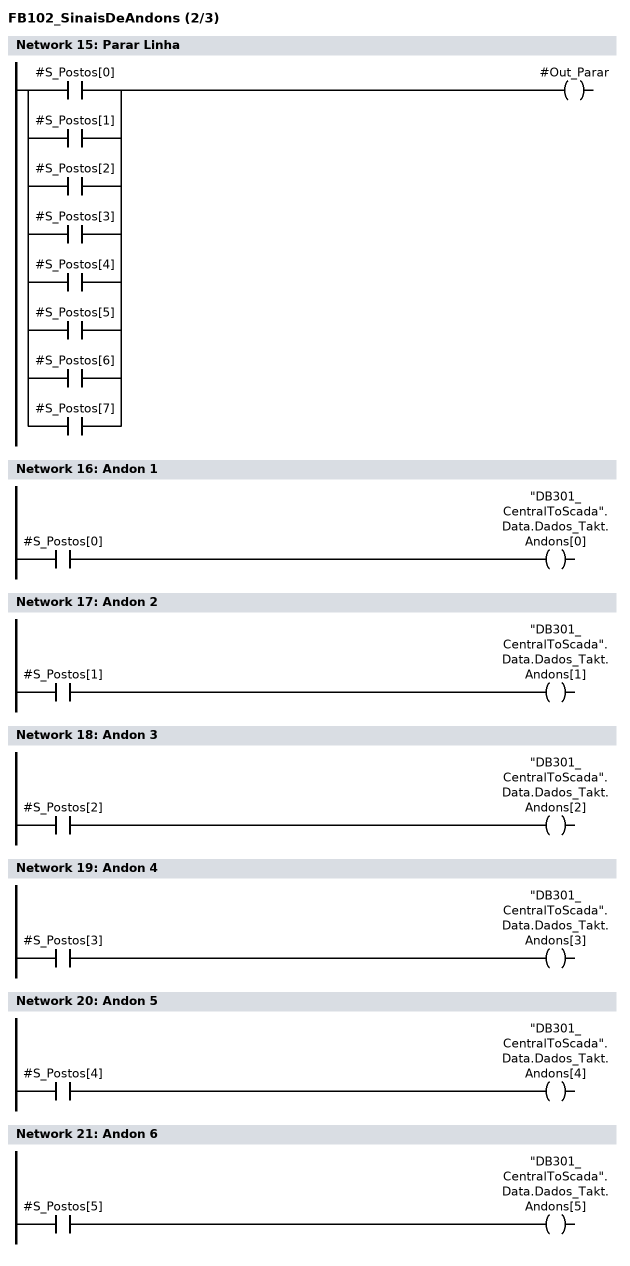
   RUNG wire#powerrail
      Contact( #S_Postos[0] )
      wire#w1
      Coil( #Out_Parar )
   END_RUNG
   RUNG wire#powerrail
      Contact( #S_Postos[1] )
   END_RUNG wire#w1
   RUNG wire#powerrail
      Contact( #S_Postos[2] )
   END_RUNG wire#w1
   RUNG wire#powerrail
      Contact( #S_Postos[3] )
   END_RUNG wire#w1
   RUNG wire#powerrail
      Contact( #S_Postos[4] )
   END_RUNG wire#w1
   RUNG wire#powerrail
      Contact( #S_Postos[5] )
   END_RUNG wire#w1
   RUNG wire#powerrail
      Contact( #S_Postos[6] )
   END_RUNG wire#w1
   RUNG wire#powerrail
      Contact( #S_Postos[7] )
   END_RUNG wire#w1
   // the same network as SCL:
   #Out_Parar := #S_Postos[0] OR #S_Postos[1] OR #S_Postos[2] OR #S_Postos[3] OR #S_Postos[4] OR #S_Postos[5] OR #S_Postos[6] OR #S_Postos[7];
END_REGION

REGION Network 16: Andon 1
   RUNG wire#powerrail
      Contact( #S_Postos[0] )
      Coil( "DB301_CentralToScada".Data.Dados_Takt.Andons[0] )
   END_RUNG
   // the same network as SCL:
   "DB301_CentralToScada".Data.Dados_Takt.Andons[0] := #S_Postos[0];
END_REGION

REGION Network 17: Andon 2
   RUNG wire#powerrail
      Contact( #S_Postos[1] )
      Coil( "DB301_CentralToScada".Data.Dados_Takt.Andons[1] )
   END_RUNG
   // the same network as SCL:
   "DB301_CentralToScada".Data.Dados_Takt.Andons[1] := #S_Postos[1];
END_REGION

REGION Network 18: Andon 3
   RUNG wire#powerrail
      Contact( #S_Postos[2] )
      Coil( "DB301_CentralToScada".Data.Dados_Takt.Andons[2] )
   END_RUNG
   // the same network as SCL:
   "DB301_CentralToScada".Data.Dados_Takt.Andons[2] := #S_Postos[2];
END_REGION

REGION Network 19: Andon 4
   RUNG wire#powerrail
      Contact( #S_Postos[3] )
      Coil( "DB301_CentralToScada".Data.Dados_Takt.Andons[3] )
   END_RUNG
   // the same network as SCL:
   "DB301_CentralToScada".Data.Dados_Takt.Andons[3] := #S_Postos[3];
END_REGION

REGION Network 20: Andon 5
   RUNG wire#powerrail
      Contact( #S_Postos[4] )
      Coil( "DB301_CentralToScada".Data.Dados_Takt.Andons[4] )
   END_RUNG
   // the same network as SCL:
   "DB301_CentralToScada".Data.Dados_Takt.Andons[4] := #S_Postos[4];
END_REGION

REGION Network 21: Andon 6
   RUNG wire#powerrail
      Contact( #S_Postos[5] )
      Coil( "DB301_CentralToScada".Data.Dados_Takt.Andons[5] )
   END_RUNG
   // the same network as SCL:
   "DB301_CentralToScada".Data.Dados_Takt.Andons[5] := #S_Postos[5];
END_REGION

REGION Network 22: Andon 7
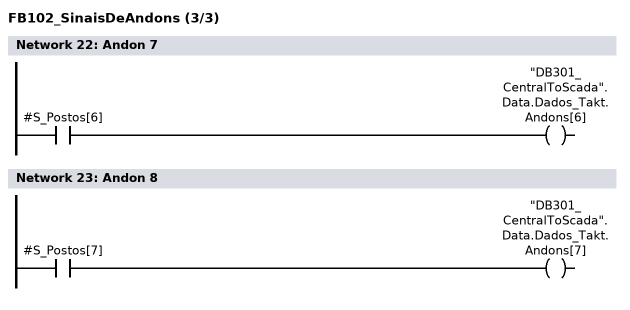
   RUNG wire#powerrail
      Contact( #S_Postos[6] )
      Coil( "DB301_CentralToScada".Data.Dados_Takt.Andons[6] )
   END_RUNG
   // the same network as SCL:
   "DB301_CentralToScada".Data.Dados_Takt.Andons[6] := #S_Postos[6];
END_REGION

REGION Network 23: Andon 8
   RUNG wire#powerrail
      Contact( #S_Postos[7] )
      Coil( "DB301_CentralToScada".Data.Dados_Takt.Andons[7] )
   END_RUNG
   // the same network as SCL:
   "DB301_CentralToScada".Data.Dados_Takt.Andons[7] := #S_Postos[7];
END_REGION
END_FUNCTION_BLOCK

FUNCTION_BLOCK "FB103_AndonsAgvs"   // FB103, LAD
TITLE = FB103_AndonsAgvs
{ S7_Optimized_Access := 'FALSE' }
VERSION : 0.1
// FB103_AndonsAgvs
   VAR_INPUT
      In_AgvEmergencia : Bool;
      In_AgvManual : Byte;
      In_AgvEmergencia_1 : Bool;
      In_AgvManual_1 : Byte;
      In_AgvEmergencia_2 : Bool;
      In_AgvManual_2 : Byte;
      In_AgvEmergencia_3 : Bool;
      In_AgvManual_3 : Byte;
      In_AgvEmergencia_4 : Bool;
      In_AgvManual_4 : Byte;
      In_AgvEmergencia_5 : Bool;
      In_AgvManual_5 : Byte;
      In_AgvEmergencia_6 : Bool;
      In_AgvManual_6 : Byte;
      In_AgvEmergencia_7 : Bool;
      In_AgvManual_7 : Byte;
   END_VAR
   VAR_OUTPUT
      Out_ParaLinha : Bool;
      Out_Emergencia : Bool;
   END_VAR
   VAR
      S_Agvs : Array[0..7] of Bool;
   END_VAR
BEGIN

REGION Network 1: AGV 1
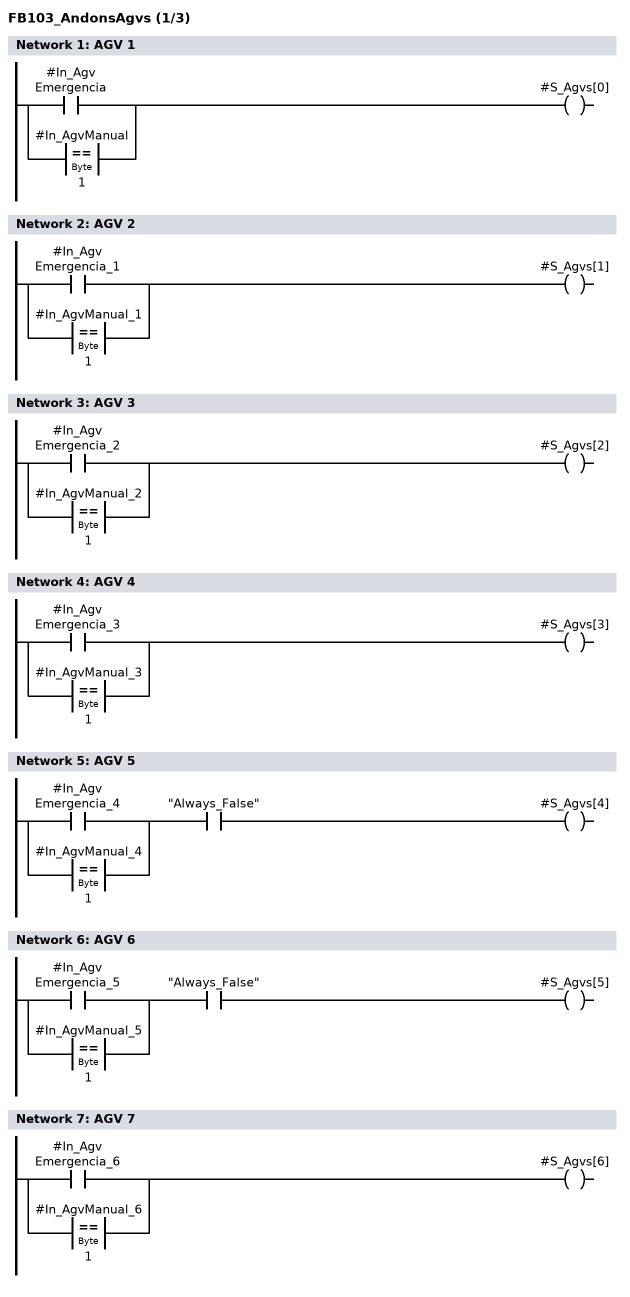
   RUNG wire#powerrail
      Contact( #In_AgvEmergencia )
      wire#w1
      Coil( #S_Agvs[0] )
   END_RUNG
   RUNG wire#powerrail
      { S7_Templates := "SrcType := Byte" } EQ_Contact(in1 := #In_AgvManual, in2 := 1)
   END_RUNG wire#w1
   // the same network as SCL:
   #S_Agvs[0] := #In_AgvEmergencia OR (#In_AgvManual = 1);
END_REGION

REGION Network 2: AGV 2
   RUNG wire#powerrail
      Contact( #In_AgvEmergencia_1 )
      wire#w1
      Coil( #S_Agvs[1] )
   END_RUNG
   RUNG wire#powerrail
      { S7_Templates := "SrcType := Byte" } EQ_Contact(in1 := #In_AgvManual_1, in2 := 1)
   END_RUNG wire#w1
   // the same network as SCL:
   #S_Agvs[1] := #In_AgvEmergencia_1 OR (#In_AgvManual_1 = 1);
END_REGION

REGION Network 3: AGV 3
   RUNG wire#powerrail
      Contact( #In_AgvEmergencia_2 )
      wire#w1
      Coil( #S_Agvs[2] )
   END_RUNG
   RUNG wire#powerrail
      { S7_Templates := "SrcType := Byte" } EQ_Contact(in1 := #In_AgvManual_2, in2 := 1)
   END_RUNG wire#w1
   // the same network as SCL:
   #S_Agvs[2] := #In_AgvEmergencia_2 OR (#In_AgvManual_2 = 1);
END_REGION

REGION Network 4: AGV 4
   RUNG wire#powerrail
      Contact( #In_AgvEmergencia_3 )
      wire#w1
      Coil( #S_Agvs[3] )
   END_RUNG
   RUNG wire#powerrail
      { S7_Templates := "SrcType := Byte" } EQ_Contact(in1 := #In_AgvManual_3, in2 := 1)
   END_RUNG wire#w1
   // the same network as SCL:
   #S_Agvs[3] := #In_AgvEmergencia_3 OR (#In_AgvManual_3 = 1);
END_REGION

REGION Network 5: AGV 5
   RUNG wire#powerrail
      Contact( #In_AgvEmergencia_4 )
      wire#w1
      Contact( "Always_False" )
      Coil( #S_Agvs[4] )
   END_RUNG
   RUNG wire#powerrail
      { S7_Templates := "SrcType := Byte" } EQ_Contact(in1 := #In_AgvManual_4, in2 := 1)
   END_RUNG wire#w1
   // the same network as SCL:
   #S_Agvs[4] := (#In_AgvEmergencia_4 OR (#In_AgvManual_4 = 1)) AND "Always_False";
END_REGION

REGION Network 6: AGV 6
   RUNG wire#powerrail
      Contact( #In_AgvEmergencia_5 )
      wire#w1
      Contact( "Always_False" )
      Coil( #S_Agvs[5] )
   END_RUNG
   RUNG wire#powerrail
      { S7_Templates := "SrcType := Byte" } EQ_Contact(in1 := #In_AgvManual_5, in2 := 1)
   END_RUNG wire#w1
   // the same network as SCL:
   #S_Agvs[5] := (#In_AgvEmergencia_5 OR (#In_AgvManual_5 = 1)) AND "Always_False";
END_REGION

REGION Network 7: AGV 7
   RUNG wire#powerrail
      Contact( #In_AgvEmergencia_6 )
      wire#w1
      Coil( #S_Agvs[6] )
   END_RUNG
   RUNG wire#powerrail
      { S7_Templates := "SrcType := Byte" } EQ_Contact(in1 := #In_AgvManual_6, in2 := 1)
   END_RUNG wire#w1
   // the same network as SCL:
   #S_Agvs[6] := #In_AgvEmergencia_6 OR (#In_AgvManual_6 = 1);
END_REGION

REGION Network 8: Para linha
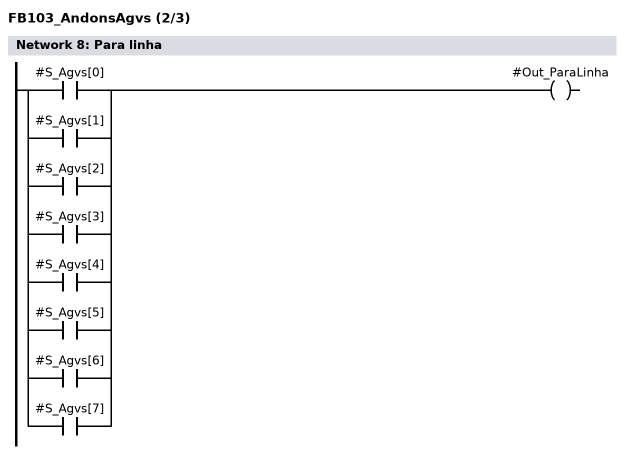
   RUNG wire#powerrail
      Contact( #S_Agvs[0] )
      wire#w1
      Coil( #Out_ParaLinha )
   END_RUNG
   RUNG wire#powerrail
      Contact( #S_Agvs[1] )
   END_RUNG wire#w1
   RUNG wire#powerrail
      Contact( #S_Agvs[2] )
   END_RUNG wire#w1
   RUNG wire#powerrail
      Contact( #S_Agvs[3] )
   END_RUNG wire#w1
   RUNG wire#powerrail
      Contact( #S_Agvs[4] )
   END_RUNG wire#w1
   RUNG wire#powerrail
      Contact( #S_Agvs[5] )
   END_RUNG wire#w1
   RUNG wire#powerrail
      Contact( #S_Agvs[6] )
   END_RUNG wire#w1
   RUNG wire#powerrail
      Contact( #S_Agvs[7] )
   END_RUNG wire#w1
   // the same network as SCL:
   #Out_ParaLinha := #S_Agvs[0] OR #S_Agvs[1] OR #S_Agvs[2] OR #S_Agvs[3] OR #S_Agvs[4] OR #S_Agvs[5] OR #S_Agvs[6] OR #S_Agvs[7];
END_REGION

REGION Network 9: Emergencia
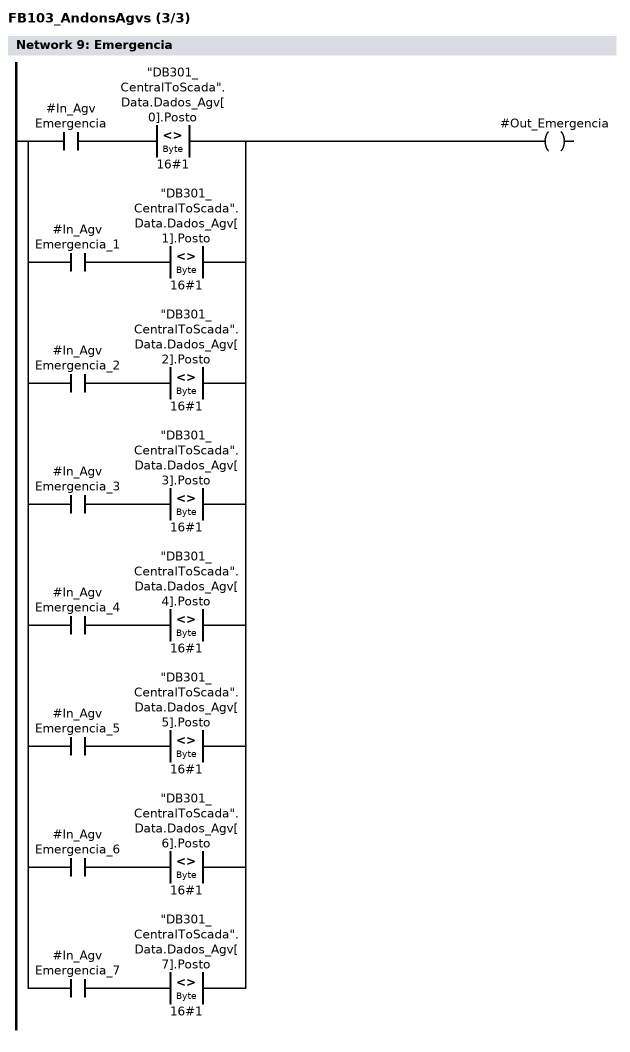
   RUNG wire#powerrail
      Contact( #In_AgvEmergencia )
      { S7_Templates := "SrcType := Byte" } NE_Contact(in1 := "DB301_CentralToScada".Data.Dados_Agv[0].Posto, in2 := 16#1)
      wire#w1
      Coil( #Out_Emergencia )
   END_RUNG
   RUNG wire#powerrail
      Contact( #In_AgvEmergencia_1 )
      { S7_Templates := "SrcType := Byte" } NE_Contact(in1 := "DB301_CentralToScada".Data.Dados_Agv[1].Posto, in2 := 16#1)
   END_RUNG wire#w1
   RUNG wire#powerrail
      Contact( #In_AgvEmergencia_2 )
      { S7_Templates := "SrcType := Byte" } NE_Contact(in1 := "DB301_CentralToScada".Data.Dados_Agv[2].Posto, in2 := 16#1)
   END_RUNG wire#w1
   RUNG wire#powerrail
      Contact( #In_AgvEmergencia_3 )
      { S7_Templates := "SrcType := Byte" } NE_Contact(in1 := "DB301_CentralToScada".Data.Dados_Agv[3].Posto, in2 := 16#1)
   END_RUNG wire#w1
   RUNG wire#powerrail
      Contact( #In_AgvEmergencia_4 )
      { S7_Templates := "SrcType := Byte" } NE_Contact(in1 := "DB301_CentralToScada".Data.Dados_Agv[4].Posto, in2 := 16#1)
   END_RUNG wire#w1
   RUNG wire#powerrail
      Contact( #In_AgvEmergencia_5 )
      { S7_Templates := "SrcType := Byte" } NE_Contact(in1 := "DB301_CentralToScada".Data.Dados_Agv[5].Posto, in2 := 16#1)
   END_RUNG wire#w1
   RUNG wire#powerrail
      Contact( #In_AgvEmergencia_6 )
      { S7_Templates := "SrcType := Byte" } NE_Contact(in1 := "DB301_CentralToScada".Data.Dados_Agv[6].Posto, in2 := 16#1)
   END_RUNG wire#w1
   RUNG wire#powerrail
      Contact( #In_AgvEmergencia_7 )
      { S7_Templates := "SrcType := Byte" } NE_Contact(in1 := "DB301_CentralToScada".Data.Dados_Agv[7].Posto, in2 := 16#1)
   END_RUNG wire#w1
   // the same network as SCL:
   #Out_Emergencia := (#In_AgvEmergencia AND ("DB301_CentralToScada".Data.Dados_Agv[0].Posto <> 16#1)) OR (#In_AgvEmergencia_1 AND ("DB301_CentralToScada".Data.Dados_Agv[1].Posto <> 16#1)) OR (#In_AgvEmergencia_2 AND ("DB301_CentralToScada".Data.Dados_Agv[2].Posto <> 16#1)) OR (#In_AgvEmergencia_3 AND ("DB301_CentralToScada".Data.Dados_Agv[3].Posto <> 16#1)) OR (#In_AgvEmergencia_4 AND ("DB301_CentralToScada".Data.Dados_Agv[4].Posto <> 16#1)) OR (#In_AgvEmergencia_5 AND ("DB301_CentralToScada".Data.Dados_Agv[5].Posto <> 16#1)) OR (#In_AgvEmergencia_6 AND ("DB301_CentralToScada".Data.Dados_Agv[6].Posto <> 16#1)) OR (#In_AgvEmergencia_7 AND ("DB301_CentralToScada".Data.Dados_Agv[7].Posto <> 16#1));
END_REGION
END_FUNCTION_BLOCK

// folder: 02_Comunicação/01_FB

FUNCTION_BLOCK "FB200_Leitura/EscritaDadosAgv"   // FB200, SCL
TITLE = FB205_Leitura/EscritaDadosAgv
{ S7_Optimized_Access := 'FALSE' }
VERSION : 0.1
// FB205_Leitura/EscritaDadosAgv
   VAR
      GET_DadosAgv1 : GET;
      PUT_DadosAgv1 : PUT;
      GET_DadosAgv2 : GET;
      PUT_DadosAgv2 : PUT;
      GET_DadosAgv3 : GET;
      PUT_DadosAgv3 : PUT;
      GET_DadosAgv4 : GET;
      PUT_DadosAgv4 : PUT;
      GET_DadosAgv5 : GET;
      PUT_DadosAgv5 : PUT;
      GET_DadosAgv6 : GET;
      PUT_DadosAgv6 : PUT;
      GET_DadosAgv7 : GET;
      PUT_DadosAgv7 : PUT;
      GET_DadosAgv8 : GET;
      PUT_DadosAgv8 : PUT;
      S_Contador : CTU;
      S_Chamada : Array[0..20] of Bool;
      S_CU : Bool;
   END_VAR
BEGIN

   REGION Contador


       #S_Contador(CU := "CM_0.1s",
                   R := #S_Chamada[13],
                   PV := 13);
   END_REGION




   CASE #S_Contador.CV OF
       0:
           #S_Chamada[13] := 0;
           #S_Chamada[0] := 1;
       1:
           #S_Chamada[0] := 0;
           #S_Chamada[1] := 1;
       2:
           #S_Chamada[1] := 0;
           #S_Chamada[2] := 1;
       3:
           #S_Chamada[2] := 0;
           #S_Chamada[3] := 1;
       4:
           #S_Chamada[3] := 0;
           #S_Chamada[4] := 1;
       5:
           #S_Chamada[4] := 0;
           #S_Chamada[5] := 1;
       6:
           #S_Chamada[5] := 0;
           #S_Chamada[6] := 1;
       7:
           #S_Chamada[6] := 0;
           #S_Chamada[7] := 1;
       8:
           #S_Chamada[7] := 0;
           #S_Chamada[8] := 1;
       9:
           #S_Chamada[8] := 0;
           #S_Chamada[9] := 1;
       10:
           #S_Chamada[9] := 0;
           #S_Chamada[10] := 1;
       11:
           #S_Chamada[10] := 0;
           #S_Chamada[11] := 1;
       12:
           #S_Chamada[11] := 0;
           #S_Chamada[12] := 1;
       13:
           #S_Chamada[12] := 0;
           #S_Chamada[13] := 1;
       ELSE
           #S_Chamada[0] := 0;
           #S_Chamada[1] := 0;
           #S_Chamada[2] := 0;
           #S_Chamada[3] := 0;
           #S_Chamada[4] := 0;
           #S_Chamada[5] := 0;
           #S_Chamada[6] := 0;
           #S_Chamada[7] := 0;
           #S_Chamada[8] := 0;
           #S_Chamada[9] := 0;
           #S_Chamada[10] := 0;

   END_CASE;







   REGION RequisiçãoDeDados
       //AGV 1
       REGION AGV1
           //Leitura do dados do AGV 1
           #GET_DadosAgv1(REQ := #S_Chamada[0],
                          ID := 16#2,
                          ADDR_1 := P# DB700.DBX0.0 BYTE 22,
                          RD_1 := P# DB301.DBX0.0 BYTE 22);
           //Escrita do dados do AGV 1
           #PUT_DadosAgv1(REQ := #S_Chamada[1],
                          ID := W#16#2,
                          ADDR_1 := P#DB701.DBX0.0 BYTE 3,
                          SD_1 := P#DB200.DBX0.0 BYTE 3);
       END_REGION
       //AGV 2
       REGION AGV2
           //Leitura do dados do AGV 2
           #GET_DadosAgv2(REQ := #S_Chamada[2] ,
                          ID := 16#3,
                          ADDR_1 := P# DB700.DBX0.0 BYTE 22,
                          RD_1 := P# DB301.DBX24.0 BYTE 22);
           //Escrita do dados do AGV 2
           #PUT_DadosAgv2(REQ := #S_Chamada[3] ,
                          ID := W#16#3,
                          ADDR_1 := P#DB701.DBX0.0 BYTE 3,
                          SD_1 := P#DB200.DBX0.0 BYTE 3);
       END_REGION
       //AGV 3
       REGION AGV3
           //Leitura do dados do AGV 3
           #GET_DadosAgv3(REQ := #S_Chamada[4] ,
                          ID := 16#4,
                          ADDR_1 := P# DB700.DBX0.0 BYTE 22,
                          RD_1 := P# DB301.DBX48.0 BYTE 22);
           //Escrita do dados do AGV 3
           #PUT_DadosAgv3(REQ := #S_Chamada[5] ,
                          ID := W#16#4,
                          ADDR_1 := P#DB701.DBX0.0 BYTE 3,
                          SD_1 := P#DB200.DBX0.0 BYTE 3);
       END_REGION
       //AGV 4
       REGION AGV4
           //Leitura do dados do AGV 4
           #GET_DadosAgv4(REQ := #S_Chamada[6] ,
                          ID := 16#5,
                         ADDR_1 := P# DB700.DBX0.0 Byte 22,
                      RD_1 := P#DB301.DBX72.0 Byte 22);
           //Escrita do dados do AGV 4
           #PUT_DadosAgv4(REQ := #S_Chamada[7] ,
                          ID := W#16#5,
                          ADDR_1 := P#DB701.DBX0.0 BYTE 3,
                          SD_1 := P#DB200.DBX0.0 BYTE 3);
       END_REGION
       //AGV 5
       REGION AGV5
           //Leitura do dados do AGV 5
           #GET_DadosAgv5(REQ := #S_Chamada[8],
                          ID := 16#6,
                          ADDR_1 := P# DB700.DBX0.0 BYTE 22,
                          RD_1 := P# DB301.DBX96.0 BYTE 22);
           //Escrita do dados do AGV 7
           #PUT_DadosAgv5(REQ := #S_Chamada[9],
                          ID := W#16#6,
                          ADDR_1 := P#DB701.DBX0.0 BYTE 3,
                          SD_1 := P#DB200.DBX0.0 BYTE 3);
       END_REGION
       //AGV 6
       REGION AGV6
           //Leitura do dados do AGV 6
           #GET_DadosAgv6(REQ := #S_Chamada[10],
                          ID := 16#7,
                          ADDR_1 := P# DB700.DBX0.0 BYTE 22,
                          RD_1 := P# DB301.DBX120.0 BYTE 22);
           //Escrita do dados do AGV 7
           #PUT_DadosAgv6(REQ := #S_Chamada[11],
                          ID := W#16#7,
                          ADDR_1 := P#DB701.DBX0.0 BYTE 3,
                          SD_1 := P#DB200.DBX0.0 BYTE 3);
       END_REGION
       //AGV 7
       REGION AGV7
           //Leitura do dados do AGV 7
           #GET_DadosAgv7(REQ := #S_Chamada[12] ,
                          ID := 16#8,
                          ADDR_1 := P# DB700.DBX0.0 BYTE 22,
                          RD_1 := P# DB301.DBX144.0 BYTE 22);
           //Escrita do dados do AGV 7
           #PUT_DadosAgv7(REQ := #S_Chamada[13] ,
                          ID := W#16#8,
                          ADDR_1 := P#DB701.DBX0.0 BYTE 3,
                          SD_1 := P#DB200.DBX0.0 BYTE 3);
       END_REGION
   END_REGION
END_FUNCTION_BLOCK

FUNCTION_BLOCK "FB201_Comunicação"   // FB201, SCL
TITLE = FB203_Comunicação
{ S7_Optimized_Access := 'FALSE' }
AUTHOR : ssbjvq
VERSION : 0.1
// FB203_Comunicação
   VAR
      S_ChamadaScada : Bool;
      S_WriteScada : Bool;
      "Leitura/EscritaDadosAgv" : "FB200_Leitura/EscritaDadosAgv";   // Bloco que concentra as requisiçoes de dados dos AGVs
      VerificaConexão_Instance : "FB202_VerificaConexão";
   END_VAR
BEGIN
   (*
   Este bloco realiza a leitura/escrita de dados no AGV e no Scada
   *)


   REGION Comunicacao_Agv
       #"Leitura/EscritaDadosAgv"();
   END_REGION

   REGION VerificaConexão_Agv
      // #VerificaConexão_Instance();
   END_REGION
END_FUNCTION_BLOCK

FUNCTION_BLOCK "FB202_VerificaConexão"   // FB202, SCL
TITLE = FB204_VerificaConexão
{ S7_Optimized_Access := 'FALSE' }
VERSION : 0.1
// Verifica Conexão com os AGVs
   VAR
      S_ConexaoAgv : Array[0..8] of Struct
         EN_R : Bool;
         ID : Word;   // Endereço do dispositivo em Rede
         RETVAL : Int;
         ERROR : Bool;
         STATUS : Word;
         C_CONN : Bool;
         C_STATUS : Word;
      END_STRUCT;
      S_Conectado : Array[0..8] of Bool;
      Counter_For : Int;
      Clock_Instance : "FB1000_Clock";
   END_VAR
   // S_ConexaoAgv[0].ID := 16#1;
   // S_ConexaoAgv[1].ID := 16#2;
   // S_ConexaoAgv[2].ID := 16#3;
   // S_ConexaoAgv[3].ID := 16#4;
   // S_ConexaoAgv[4].ID := 16#5;
   // S_ConexaoAgv[5].ID := 16#6;
   // S_ConexaoAgv[6].ID := 16#7;
   // S_ConexaoAgv[7].ID := 16#8;
   // S_ConexaoAgv[8].ID := 16#9;
   // // S_ConexaoAgv[0] : Conexão Scada/Plc IT
   // // S_ConexaoAgv[1] : Conexão AGV 1
   // // S_ConexaoAgv[2] : Conexão AGV 2
   // // S_ConexaoAgv[3] : Conexão AGV 3
   // // S_ConexaoAgv[4] : Conexão AGV 4
   // // S_ConexaoAgv[5] : Conexão AGV 5
   // // S_ConexaoAgv[6] : Conexão AGV 6
   // // S_ConexaoAgv[7] : Conexão AGV 7
   // // S_ConexaoAgv[8] : Conexão AGV 8
BEGIN

   REGION Verifica_Status_Conexao
       #Clock_Instance(In_Tempo := T#10s);
       IF #Clock_Instance.Out_Sinal THEN
           FOR #Counter_For := 1 TO 9 DO
               //Verifica se os AGVs/Scada estão conectados
               C_CNTRL(EN_R := #S_ConexaoAgv[#Counter_For].EN_R,
                       ID := #S_ConexaoAgv[#Counter_For].ID,
                       RETVAL => #S_ConexaoAgv[#Counter_For].RETVAL,
                       ERROR => #S_ConexaoAgv[#Counter_For].ERROR,
                       STATUS => #S_ConexaoAgv[#Counter_For].STATUS,
                       C_CONN => #S_ConexaoAgv[#Counter_For].C_CONN,
                       C_STATUS => #S_ConexaoAgv[#Counter_For].C_STATUS);
               //Se conectado seta uma memoria
               IF #S_ConexaoAgv[#Counter_For].C_CONN THEN
                   #S_Conectado[#Counter_For] := 1;
               ELSE
                   #S_Conectado[#Counter_For] := 0;
               END_IF;

           END_FOR;
       END_IF;

   END_REGION
END_FUNCTION_BLOCK

// folder: 04_Services/01_FB

FUNCTION_BLOCK "FB1000_Clock"   // FB1000, LAD
TITLE = FB1000_Clock
{ S7_Optimized_Access := 'FALSE' }
VERSION : 0.1
// FB1000_Clock
   VAR_INPUT
      In_Tempo : Time;
   END_VAR
   VAR_OUTPUT
      Out_Sinal : Bool;
      Out_NotSinal : Bool;
   END_VAR
   VAR
      TON_1 : TON;
      TON_2 : TON;
   END_VAR
BEGIN

REGION Network 1
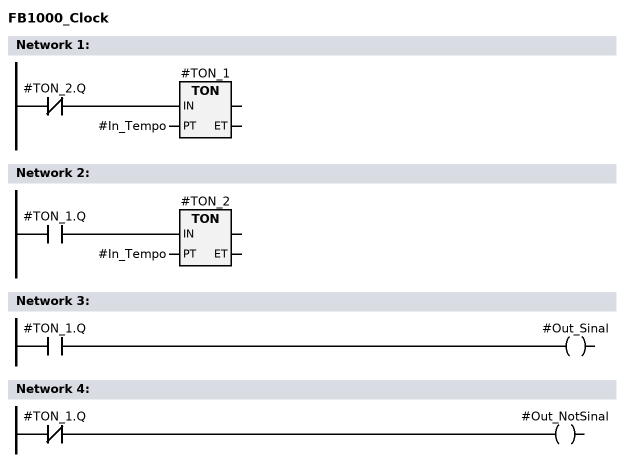
   #TON_1.TON(IN := NOT #TON_2.Q, PT := #In_Tempo);
END_REGION

REGION Network 2
   #TON_2.TON(IN := #TON_1.Q, PT := #In_Tempo);
END_REGION

REGION Network 3
   RUNG wire#powerrail
      Contact( #TON_1.Q )
      Coil( #Out_Sinal )
   END_RUNG
   // the same network as SCL:
   #Out_Sinal := #TON_1.Q;
END_REGION

REGION Network 4
   RUNG wire#powerrail
      I_Contact( #TON_1.Q )
      Coil( #Out_NotSinal )
   END_RUNG
   // the same network as SCL:
   #Out_NotSinal := NOT #TON_1.Q;
END_REGION
END_FUNCTION_BLOCK